// TwinCAT 3 PLC project fridge1
// ProgramVersion: 3.1.4026.21
// CompilerDefines: VISU_USEPROPERTYINFO
// libraries:
//   Tc2_Standard, * (Beckhoff Automation GmbH)
//   Tc2_System, * (Beckhoff Automation GmbH)
//   VisuSymbols, 4.5.0.0 (System)
// project tree:
//   / GlobalTextList.TcGTLO, PlcTask.TcTTO, Visualization Manager.TcVMO (not stored), VisuMain.TcVIS
//   GVLs/ GVL_Var.TcGVL
//   POUs/ Fridge2.TcPOU, Fridge1.TcPOU, Fridge2B.TcPOU, Fridge3A.TcPOU, Fridge3B.TcPOU, TemperatureSimulator.TcPOU
// real-time tasks:
//   TASK PlcTask: cycle T#10ms, priority 20, ADS port 350

CONFIGURATION fridge1
    RESOURCE PLC ON TwinCAT3
        TASK PlcTask(INTERVAL := T#10ms, PRIORITY := 20);
        PROGRAM Fridge3A WITH PlcTask : Fridge3A;
        PROGRAM TemperatureSimulator WITH PlcTask : TemperatureSimulator;
    END_RESOURCE
END_CONFIGURATION

// ---- GVLs/GVL_Var.TcGVL
{attribute 'qualified_only'}
VAR_GLOBAL
	bDoorOpen : BOOL; // to set the door open
	bAlarmReset : BOOL; // TRUE = door open, button to reset alarm
	fTempActual : REAL := 5.0; // Actual temperature
	fTempSet : REAL := 8.0; // Set temperature
	fHysteresis : REAL := 1.0;
	// Outputs
	bLight : BOOL; // Interior light
	bAlarmOut : BOOL;
	
	bCompressor : BOOL := FALSE; // Compressor state (init OFF)
	bCompressure: BOOL;
END_VAR

// ---- POUs/Fridge3A.TcPOU
PROGRAM Fridge3A
VAR
// Inputs (simulated)
	
	
	
	

	
	tDoorOpenThreshold : TIME := T#10S; //Time from door opening after which alarm turns on
	
	fbTimerDoorAlarm : TON;
	bAlarmLatched : BOOL; // Latched alaram state
END_VAR

// Light control (same as before)
GVL_Var.bLight := GVL_Var.bDoorOpen;
// Door alarm timer
fbTimerDoorAlarm(IN := GVL_Var.bDoorOpen, PT := tDoorOpenThreshold);
// Alarm logic with latching
IF fbTimerDoorAlarm.Q THEN
	bAlarmLatched := TRUE;
END_IF
// Reset alarm
IF GVL_Var.bAlarmReset THEN
	bAlarmLatched := FALSE;
END_IF
// Output alarm
GVL_Var.bAlarmOut := bAlarmLatched;
// Compressor control
IF GVL_Var.fTempActual > GVL_Var.fTempSet THEN
	GVL_Var.bCompressor := TRUE; // Warm: turn ON
ELSE
	GVL_Var.bCompressor := FALSE; // Cold: turn OFF
END_IF

END_PROGRAM

// ---- POUs/TemperatureSimulator.TcPOU
PROGRAM TemperatureSimulator
VAR
	fbT1 : TON;
	//The temperature is decreased on a time delay, when the compressor has been activated
	tCooling : TIME := T#500MS;
	bReduceTemp : BOOL; //Signal for decreasing the temperature
	fbT2 : TON;
	// The temperature is increased on a time delay, when the compressor is off
	tEnvironment : TIME := T#2S; //Delay time when the door is closed
	tEnvironmentDoorOpen : TIME := T#1S; //Delay time when the door is open
	bRaiseTemp : BOOL; //Signal for increasing the temperature
	tImTemp : TIME; //Delay time for warning due to environment
	nCounter : INT;
	Visualization: INT;
	HMI: INT;
END_VAR

IF GVL_Var.fTempActual > (GVL_Var.fTempSet+GVL_Var.fHysteresis) THEN
GVL_Var.bCompressure := TRUE;
END_IF

IF GVL_Var.fTempActual < (GVL_Var.fTempSet-GVL_Var.fHysteresis) THEN
GVL_Var.bCompressure := FALSE;
END_IF


(* Normal warming process: interaction with the environment *)
//If the door is open, warming will occur faster; SEL selects tEnvironmentDoorOpen
tImTemp:=SEL(GVL_Var.bDoorOpen, tEnvironment, tEnvironmentDoorOpen);
//The temperature is incremented by 0.1°C per cycle after a delay of tImTemp
fbT2(IN:= TRUE, PT:= tImTemp, Q=>bRaiseTemp);
IF bRaiseTemp THEN
		GVL_Var.fTempActual := GVL_Var.fTempActual + 0.1;
		fbT2(IN:=FALSE);
END_IF
nCounter := nCounter+1; // No function, just for showing that time is running.

END_PROGRAM

// ---- POUs/Fridge2.TcPOU
PROGRAM Fridge2
VAR
// Inputs (simulated)
	bDoorOpen : BOOL; // TRUE = door open
// Outputs
	bLight : BOOL; // Interior light
	bAlarmOut : BOOL;
	tDoorOpenThreshold : TIME := T#10S; //Time from door opening after which alarm turns on
	fbTimerDoorAlarm : TON;
END_VAR

bLight := bDoorOpen;
// Door alarm timer
fbTimerDoorAlarm(IN := bDoorOpen, PT := tDoorOpenThreshold);
// Alarm depends on timer output
bAlarmOut := fbTimerDoorAlarm.Q;

END_PROGRAM

// ---- POUs/Fridge1.TcPOU
PROGRAM Fridge1
VAR
// Inputs (simulated)
	bDoorOpen : BOOL; // TRUE = door open
// Outputs
	bLight : BOOL; // Interior light
	nCounter : INT;
END_VAR
// Simple logic: light follows door state

bLight := bDoorOpen;
nCounter := nCounter + 1;

END_PROGRAM

// ---- POUs/Fridge2B.TcPOU
PROGRAM Fridge2B
VAR
// Inputs (simulated)
	bDoorOpen : BOOL;
	bAlarmReset : BOOL; // TRUE = door open
// Outputs
	bLight : BOOL; // Interior light
	bAlarmOut : BOOL;
	tDoorOpenThreshold : TIME := T#10S; //Time from door opening after which alarm turns on
	fbTimerDoorAlarm : TON;
	bAlarmLatched : BOOL; // Latched alaram state
END_VAR

// Light control (same as before)
bLight := bDoorOpen;
// Door alarm timer
fbTimerDoorAlarm(IN := bDoorOpen, PT := tDoorOpenThreshold);
// Alarm logic with latching
IF fbTimerDoorAlarm.Q THEN
	bAlarmLatched := TRUE;
END_IF
// Reset alarm
IF bAlarmReset THEN
	bAlarmLatched := FALSE;
END_IF
// Output alarm
bAlarmOut := bAlarmLatched;

END_PROGRAM

// ---- POUs/Fridge3B.TcPOU
PROGRAM Fridge3B
VAR
// Inputs (simulated)
	
	
	
	

	
	tDoorOpenThreshold : TIME := T#10S; //Time from door opening after which alarm turns on
	
	fbTimerDoorAlarm : TON;
	bAlarmLatched : BOOL; // Latched alaram state
END_VAR

// Light control (same as before)
GVL_Var.bLight := GVL_Var.bDoorOpen;
// Door alarm timer
fbTimerDoorAlarm(IN := GVL_Var.bDoorOpen, PT := tDoorOpenThreshold);
// Alarm logic with latching
IF fbTimerDoorAlarm.Q THEN
	bAlarmLatched := TRUE;
END_IF
// Reset alarm
IF GVL_Var.bAlarmReset THEN
	bAlarmLatched := FALSE;
END_IF
// Output alarm
GVL_Var.bAlarmOut := bAlarmLatched;
// Compressor control
IF GVL_Var.fTempActual > GVL_Var.fTempSet THEN
	GVL_Var.bCompressor := TRUE; // Warm: turn ON
ELSE
	GVL_Var.bCompressor := FALSE; // Cold: turn OFF
END_IF

END_PROGRAM

// ---- GlobalTextList.TcGTLO
TEXTLIST GlobalTextList
  499 = '%.0f'
  461 = 'Alarm Door'
  634 = 'Alarm Reset'
  777 = 'Controller '
  736 = 'Monitor'
  131 = 'Monitorl'
END_TEXTLIST

// ---- VisuMain.TcVIS
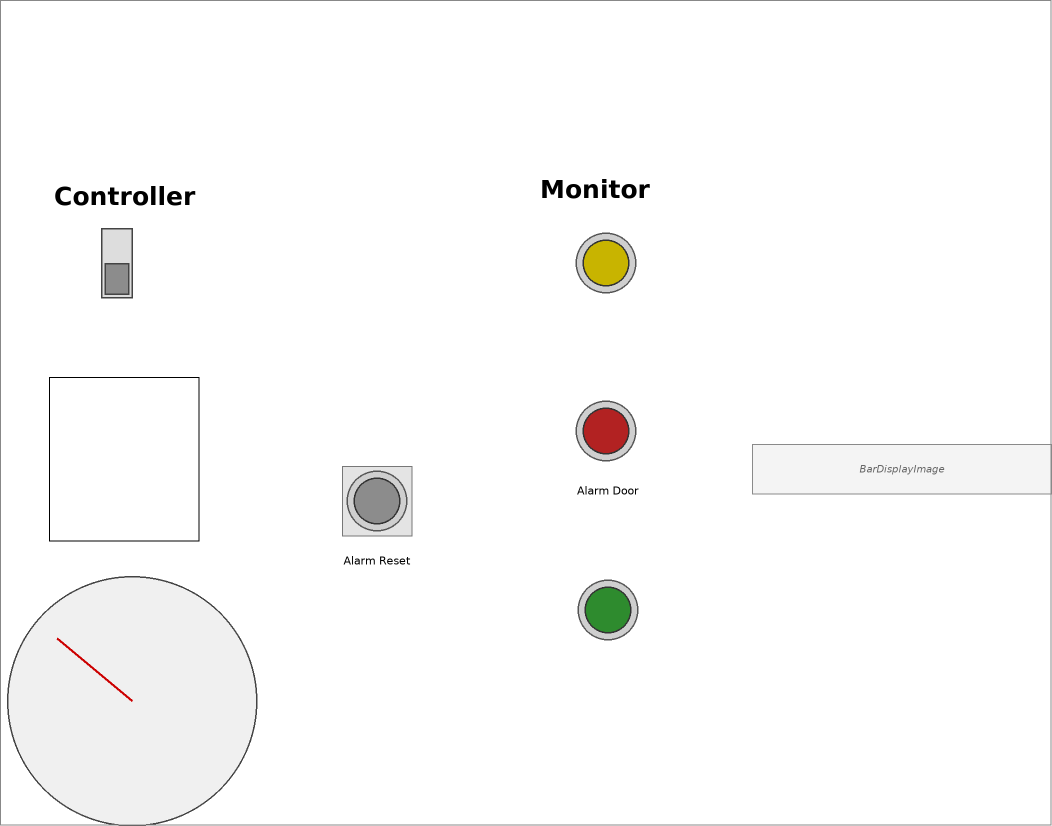
VISUALIZATION VisuMain  // 1052x826
    Lamp1 (571,228 70x70), variable: GVL_Var.bLight, style: Lamp-Lamp1-Yellow
    DipSwitch (82,228 70x70), variable: GVL_Var.bDoorOpen, behaviour: TOGGLE, style: Switch-DipSwitch-Gray
    Rectangle (49,377 150x164)
        toggle GVL_Var.bDoorOpen
    Lamp1 (571,396 70x70), variable: GVL_Var.bAlarmOut, style: Lamp-Lamp1-Red
    Label (533,476 150x30), "Alarm Door"
    Label (27,163 204x66), "Controller"
    Label (520,174 150x30), "Monitor"
    PushSwitch (342,466 70x70), variable: GVL_Var.bAlarmReset, behaviour: TOGGLE, style: Switch-PushSwitch-Gray
    Label (302,546 150x30), "Alarm Reset"
    Meter360 (7,576 250x250), value: GVL_Var.fTempSet, style: Meter-Meter360-Gray, scale format: %.0f, scale 0..20
    Lamp1 (573,575 70x70), variable: GVL_Var.bCompressor, style: Lamp-Lamp1-Green
    BarDisplayImage (752,444 300x50), value: GVL_Var.fTempActual, style: BarDisplayImage-Gray, scale format: %.1f, scale 0..24
END_VISUALIZATION
